Omron CX-Programmer project NewProject (CX-Programmer 9.73)

# PLC NewPLC1: CP1E N60

## Global symbols (name address type ; comment)
100.00 BOOL  ; Out1
W0.00 BOOL  ; PB_1

## Program NewProgram1 (cyclic task 0)

### Section Section1

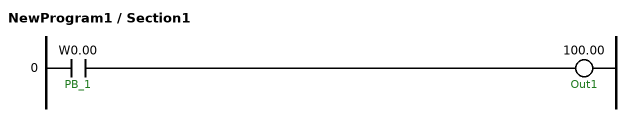
; rung 0
LD W0.00  ; PB_1
OUT 100.00  ; Out1

### Section END
; rung 0
END(001)